FUNCTION VecMulNum : Vec3
VAR_INPUT
	v : Vec3;
	n : LREAL;
END_VAR
VAR
	i : INT;
END_VAR

FOR i := 0 TO 2 DO
    VecMulNum.data[i] := n * v.data[i]; 
END_FOR

END_FUNCTION

(* stored: Version 1.1.0.1, ProductVersion 3.1.4024.2
   POU VecMulNum: Id {88fabd67-1c26-431b-b752-a955f9bdfd4b}, SpecialFunc None *)
